// Cyclic live status plus the first-out diagnostic (S3.12, S6.9).
TYPE ST_SeparatorOutImm :
STRUCT
    CarrierAt    : BOOL;
    CarrierAfter : BOOL;
    OpenedFb     : BOOL;
    ValveOpen    : BOOL;
END_STRUCT
END_TYPE

(* stored: Version 1.1.0.1, ProductVersion 3.1.4024.12
   DUT ST_SeparatorOutImm: Id {29d2faa0-5acc-456f-ba8a-7826df49373d} *)
